FUNCTION_BLOCK TcoUrRoboticsTest EXTENDS TcoUrRobotics.TcoUrCb3_v_3_x_x
VAR
    _serviceModeCount : ULINT;
    _serviceModeOverride : LREAL;
END_VAR
VAR
   
END_VAR

//SUPER^(	inEnable 			:=	inEnable,
//		inEnablePositive	:=	inEnablePositive,
//		inEnableNegative	:=	inEnableNegative,
//		inCalibrationCam	:=	inCalibrationCam,
//		inoAxisRef			:=	inoAxisRef);
//

END_FUNCTION_BLOCK

(* stored: Version 1.1.0.1, ProductVersion 3.1.4024.12
   POU TcoUrRoboticsTest: Id {3c7a463b-64d6-0aa6-14bf-e8aa4da5975e}, SpecialFunc None *)
